Staubli VAL3: S2S.dtx

bool bConnected
num nLocalTSAP_HI
num nLocalTSAP_LO
num nRemoteTSAP_HI
num nRemoteTSAP_LO
num nConnType
public num nLastError
num nPDULength
num nRecvTimeout = 0.5
sio sTCPclient
num nISOPort = 102
num nISO_CR[22]
  [0] = 3
  [3] = 22
  [4] = 17
  [5] = 224
  [9] = 1
  [11] = 192
  [12] = 1
  [13] = 10
  [14] = 193
  [15] = 2
  [16] = 1
  [18] = 194
  [19] = 2
  [20] = 1
  [21] = 2
num nErrISOConnFail = 6
num nLastPDUType
num nCC = 208
num nErrISOInvPDU = 8
num nErrTCPConnRst = 2
num nMaxPduSize = 247
num nMinPduSize = 16
num nISOheaderSize = 7
num nWRsize = 35
num nDataSize
num nShift = 17
num nS7_PN[25]
  [0] = 3
  [3] = 25
  [4] = 2
  [5] = 240
  [6] = 128
  [7] = 50
  [8] = 1
  [11] = 4
  [14] = 8
  [17] = 240
  [20] = 1
  [22] = 1
  [24] = 240
num nErrISONegPDU = 7
num nTempBuffer
public num nAreaPE = 129
public num nAreaPA = 130
public num nAreaMK = 131
public num nAreaDB = 132
public num nAreaCT = 28
public num nAreaTM = 29
public num nNoErrors
num nS7_W[35]
  [0] = 3
  [3] = 31
  [4] = 2
  [5] = 240
  [6] = 128
  [7] = 50
  [8] = 1
  [11] = 5
  [14] = 14
  [17] = 4
  [18] = 1
  [19] = 18
  [20] = 10
  [21] = 16
  [22] = 2
  [27] = 132
  [32] = 4
num nRDsize = 31
num nWLbit = 1
num nWLbyte = 2
num nWLword = 4
num nWLdword = 6
num nWLreal = 8
num nWLcounter = 28
num nWLtimer = 29
num nErrTCPSend = 4
num nErrDataRead = 768
ISO_PDU_DATA_T PDU
  [0]
    num TPKT[4]
    num COPT[3]
    S7telegram_T S7telegram
      [0]
        num H[18]
        num DATA[240]
num nDataBuffer[500]
num nS7_R[31]
  [0] = 3
  [3] = 31
  [4] = 2
  [5] = 240
  [6] = 128
  [7] = 50
  [8] = 1
  [11] = 5
  [14] = 14
  [17] = 4
  [18] = 1
  [19] = 18
  [20] = 10
  [21] = 16
  [22] = 2
  [27] = 132
num nS7WLCounter = 28
num nS7WLTimer = 29
num nErrDataWrite = 1024
num nS7_BI[37]
  [0] = 3
  [3] = 37
  [4] = 2
  [5] = 240
  [6] = 128
  [7] = 50
  [8] = 7
  [11] = 5
  [14] = 8
  [16] = 12
  [18] = 1
  [19] = 18
  [20] = 4
  [21] = 17
  [22] = 67
  [23] = 3
  [25] = 255
  [26] = 9
  [28] = 8
  [29] = 48
  [30] = 65
  [31] = 48
  [32] = 48
  [33] = 48
  [34] = 48
  [35] = 48
  [36] = 65
num nErrS7Func = 1280
string sVersion = ""0.1.0""
